Omron CX-Programmer project NewProject (CX-Programmer 9.54)

# PLC Automation_project_Station2: CJ1M CPU11

## Global symbols (name address type ; comment)
0.00 BOOL  ; Start_PB
0.01 BOOL  ; Stop_PB
0.02 BOOL  ; Reset_PB
0.03 BOOL  ; Emergency_PB
0.04 BOOL  ; Pusher 2 Front Limit
0.05 BOOL  ; Machining_Busy
0.06 BOOL  ; Machining_Error
0.07 BOOL  ; Machining_Opened
0.08 BOOL  ; Machining_Progress
0.09 BOOL  ; Vision 2
0.10 BOOL  ; Diff_Sensor2
1.00 BOOL  ; Raw Metal Emitter
1.01 BOOL  ; Machining_Start
1.04 BOOL  ; Pusher 2
1.05 BOOL  ; Painted Base Emitter
1.06 BOOL  ; Base Machining Conveyor
1.07 BOOL  ; Base Project Conveyor
1.08 BOOL  ; Right_Tranfer Conveyor
1.09 BOOL  ; Forward_Transfer Conveyor
1.10 BOOL  ; Painting Conveyor 1
1.11 BOOL  ; Painting Conveyor 2
1.12 BOOL  ; Painting Conveyor 3
1.13 BOOL  ; Start_Light
1.14 BOOL  ; Stop_Light
1.15 BOOL  ; Reset_Light
D10 CHANNEL  ; Painted Metal Counting
D11 CHANNEL  ; Reject Counting
W10.00 BOOL  ; Right_Tranfer Conveyor_Control
W10.01 BOOL  ; Forward_Tranfer Conveyor_Control
W10.02 BOOL  ; Pusher Control
W10.03 BOOL  ; Painted Emitter Control
W10.04 BOOL  ; Reset Counting
W11.00 BOOL  ; Counting_Control_Painted
W11.01 BOOL  ; Counting_Control_Reject
W1.00 BOOL  ; Status
W1.01 BOOL  ; Emergency_Status
W20.00 BOOL  ; Machining_Busy_Status
W20.01 BOOL  ; Machining_Error_Status
W20.02 BOOL  ; Machining_Opened_Status
W20.03 BOOL  ; Machining_Progress_Status

## Program NewProgram1 (cyclic task 0)

### Section Station2

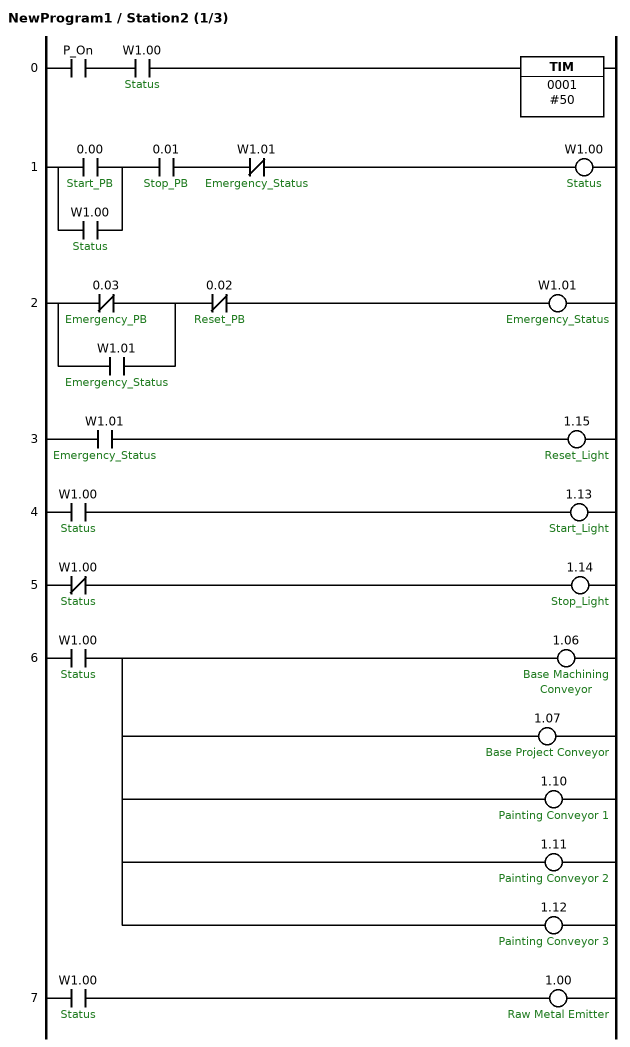
; rung 0
LD P_On
AND W1.00  ; Status
TIM 0001 #50
; rung 1
LD 0.00  ; Start_PB
OR W1.00  ; Status
AND 0.01  ; Stop_PB
ANDNOT W1.01  ; Emergency_Status
OUT W1.00  ; Status
; rung 2
LDNOT 0.03  ; Emergency_PB
OR W1.01  ; Emergency_Status
ANDNOT 0.02  ; Reset_PB
OUT W1.01  ; Emergency_Status
; rung 3
LD W1.01  ; Emergency_Status
OUT 1.15  ; Reset_Light
; rung 4
LD W1.00  ; Status
OUT 1.13  ; Start_Light
; rung 5
LDNOT W1.00  ; Status
OUT 1.14  ; Stop_Light
; rung 6
LD W1.00  ; Status
OUT 1.06  ; Base Machining Conveyor
OUT 1.07  ; Base Project Conveyor
OUT 1.10  ; Painting Conveyor 1
OUT 1.11  ; Painting Conveyor 2
OUT 1.12  ; Painting Conveyor 3
; rung 7
LD W1.00  ; Status
OUT 1.00  ; Raw Metal Emitter

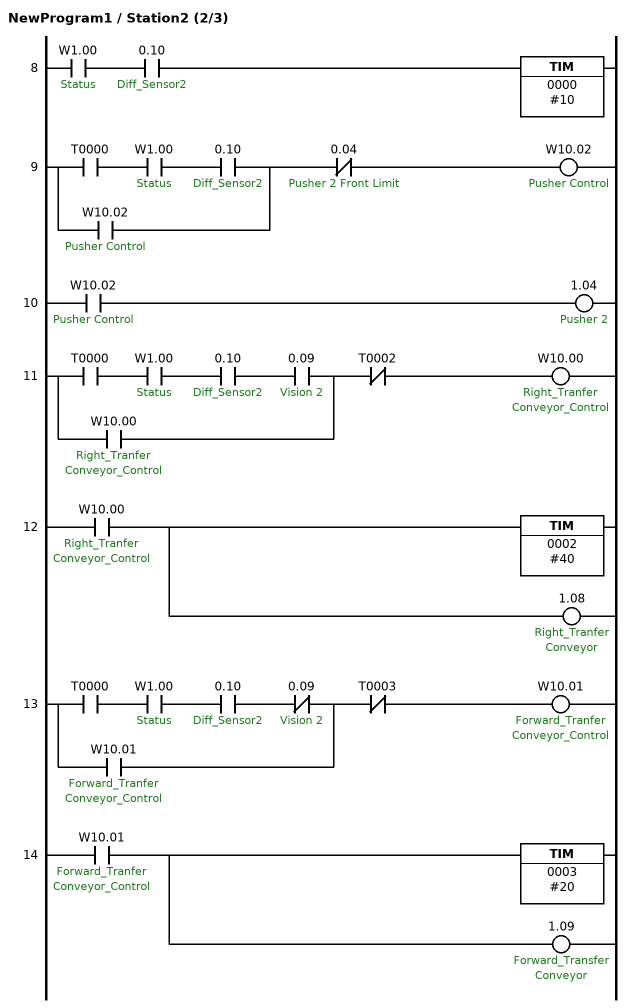
; rung 8
LD W1.00  ; Status
AND 0.10  ; Diff_Sensor2
TIM 0000 #10
; rung 9
LD T0000
AND W1.00  ; Status
AND 0.10  ; Diff_Sensor2
OR W10.02  ; Pusher Control
ANDNOT 0.04  ; Pusher 2 Front Limit
OUT W10.02  ; Pusher Control
; rung 10
LD W10.02  ; Pusher Control
OUT 1.04  ; Pusher 2
; rung 11
LD T0000
AND W1.00  ; Status
AND 0.10  ; Diff_Sensor2
AND 0.09  ; Vision 2
OR W10.00  ; Right_Tranfer Conveyor_Control
ANDNOT T0002
OUT W10.00  ; Right_Tranfer Conveyor_Control
; rung 12
LD W10.00  ; Right_Tranfer Conveyor_Control
TIM 0002 #40
OUT 1.08  ; Right_Tranfer Conveyor
; rung 13
LD T0000
AND W1.00  ; Status
AND 0.10  ; Diff_Sensor2
ANDNOT 0.09  ; Vision 2
OR W10.01  ; Forward_Tranfer Conveyor_Control
ANDNOT T0003
OUT W10.01  ; Forward_Tranfer Conveyor_Control
; rung 14
LD W10.01  ; Forward_Tranfer Conveyor_Control
TIM 0003 #20
OUT 1.09  ; Forward_Transfer Conveyor

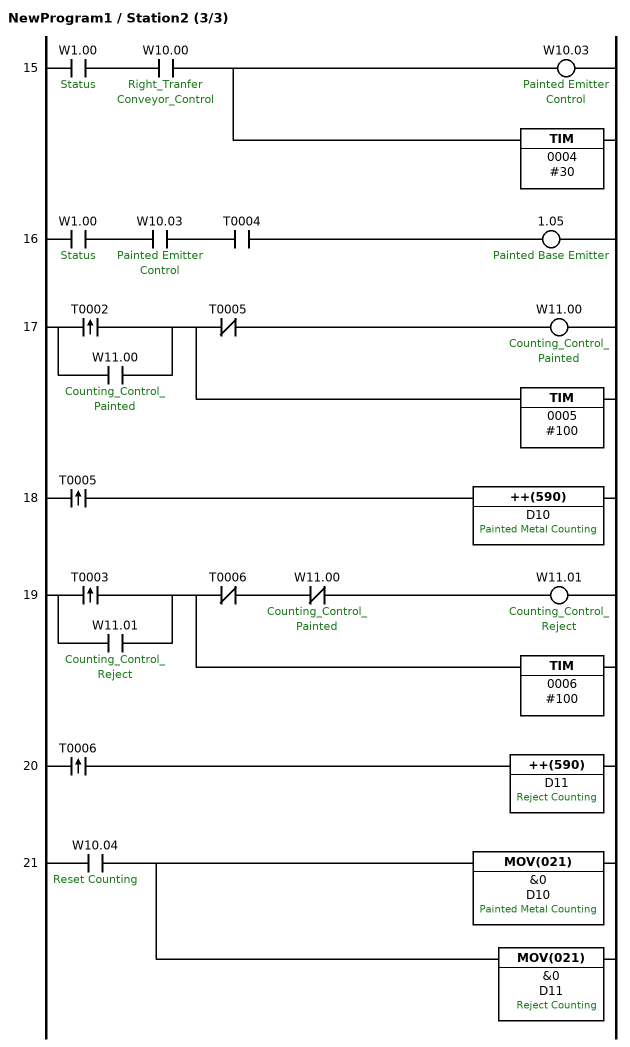
; rung 15
LD W1.00  ; Status
AND W10.00  ; Right_Tranfer Conveyor_Control
OUT W10.03  ; Painted Emitter Control
TIM 0004 #30
; rung 16
LD W1.00  ; Status
AND W10.03  ; Painted Emitter Control
AND T0004
OUT 1.05  ; Painted Base Emitter
; rung 17
@LD T0002
OR W11.00  ; Counting_Control_Painted
OUT TR0
ANDNOT T0005
OUT W11.00  ; Counting_Control_Painted
LD TR0
TIM 0005 #100
; rung 18
@LD T0005
++(590) D10  ; Painted Metal Counting
; rung 19
@LD T0003
OR W11.01  ; Counting_Control_Reject
OUT TR0
ANDNOT T0006
ANDNOT W11.00  ; Counting_Control_Painted
OUT W11.01  ; Counting_Control_Reject
LD TR0
TIM 0006 #100
; rung 20
@LD T0006
++(590) D11  ; Reject Counting
; rung 21
LD W10.04  ; Reset Counting
MOV(021) &0 D10  ; Painted Metal Counting
MOV(021) &0 D11  ; Reject Counting

### Section Base_Machining_Control

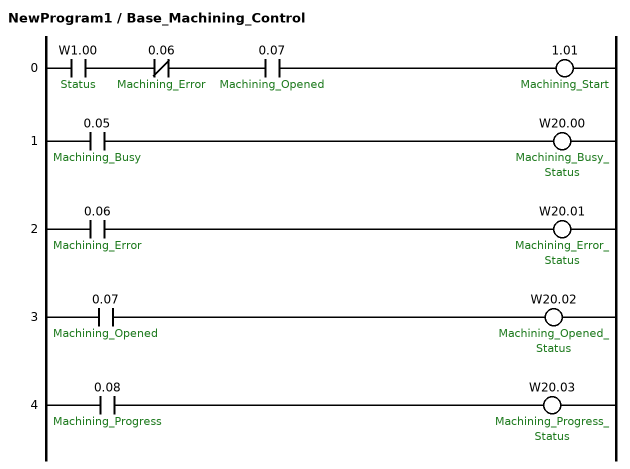
; rung 0
LD W1.00  ; Status
ANDNOT 0.06  ; Machining_Error
AND 0.07  ; Machining_Opened
OUT 1.01  ; Machining_Start
; rung 1
LD 0.05  ; Machining_Busy
OUT W20.00  ; Machining_Busy_Status
; rung 2
LD 0.06  ; Machining_Error
OUT W20.01  ; Machining_Error_Status
; rung 3
LD 0.07  ; Machining_Opened
OUT W20.02  ; Machining_Opened_Status
; rung 4
LD 0.08  ; Machining_Progress
OUT W20.03  ; Machining_Progress_Status

### Section END
; rung 0
END(001)